// TwinCAT 3 PLC project Example
// ProgramVersion: 3.1.4022.7
// libraries:
//   LCLS Vacuum, * (SLAC - LCLS)
//   LCLSVacuumSerialDriverLib, * (SLAC - LCLS)
//   Tc2_SerialCom, * (Beckhoff Automation GmbH)
//   Tc2_Standard, * (Beckhoff Automation GmbH)
//   Tc2_System, * (Beckhoff Automation GmbH)
//   Tc3_Module, * (Beckhoff Automation GmbH)
// project tree:
//   / CommTask.TcTTO, PlcTask.TcTTO
//   GVLs/ GVL_COM.TcGVL (not stored), GVL_Devices.TcGVL
//   POUs/ MAIN.TcPOU, PRG_COM.TcPOU
// real-time tasks:
//   TASK PlcTask: cycle T#10ms, priority 20, ADS port 350
//   TASK CommTask: cycle T#10ms, priority 21, ADS port 351

CONFIGURATION Example
    RESOURCE PLC ON TwinCAT3
        TASK CommTask(INTERVAL := T#10ms, PRIORITY := 21);
        TASK PlcTask(INTERVAL := T#10ms, PRIORITY := 20);
        PROGRAM PRG_COM WITH CommTask : PRG_COM;
        PROGRAM MAIN WITH PlcTask : MAIN;
    END_RESOURCE
END_CONFIGURATION

// ---- GVLs/GVL_Devices.TcGVL
VAR_GLOBAL
	
	(*TD20*)
	{attribute 'pytmc' := '
    pv: PTM:01
	'}
	PTM_01 : FB_PTM_TurboDrive; // PLC IO Interface
	PTM_01_Serial : FB_Oerlikon_TD20_COM; //Serial Interface
	
	
	(*Pfeiffer*)
	{attribute 'pytmc' := '
    pv: PTM:02
	'}
	PTM_02 : FB_PTM_Pfeiffer;
	{attribute 'pytmc' := '
    pv: PTM:03
	'}
	PTM_03 : FB_PTM_Pfeiffer;
	// They share the same serial port
	st_Pfeiffer_CTRL 			: ARRAY[1..20] OF ST_PfeifferControl;
	st_Pfeiffer_RBK 			: ARRAY[1..20] OF ST_PfeifferStatus;
	fb_PfeifferCom : FB_PFEIFFER_COM;
	
END_VAR

// ---- POUs/PRG_COM.TcPOU
PROGRAM PRG_COM
VAR
END_VAR

//needs to run on a seperate task
//PTM_01
(*Instanitate Serial port com function *) 
fbSerialLineControl(
	Mode:= SERIALLINEMODE_EL6_22B,
	pComIn:= ADR(stComIn),
	pComOut:=ADR(stComOut),
	SizeComIn:= SIZEOF(stComIn),
	TxBuffer:= SerialTXBuffer,
	RxBuffer:= SerialRXBuffer,
	Error=> ,
	ErrorID=> );
	

//PTM_02 and PTM_03
(*Instanitate Serial port com function *) 
E2_fbSerialLineControl(
	Mode:= SERIALLINEMODE_EL6_22B,
	pComIn:= ADR(E2_stComIn),
	pComOut:=ADR(E2_stComOut),
	SizeComIn:= SIZEOF(E2_stComIn),
	TxBuffer:= E2_SerialTXBuffer,
	RxBuffer:= E2_SerialRXBuffer,
	Error=> ,
	ErrorID=> );

END_PROGRAM

// ---- POUs/MAIN.TcPOU
PROGRAM MAIN
VAR
END_VAR

	
PRG_COM();

// Leybold Turbo Drive
(* Instanitate the Function block for Pump Control*)
PTM_01(i_xExtILKOk:= TRUE , iq_stPtm=> );
(* Instanitate the Function block for serial communication with TD20 *)
PTM_01_Serial(SerialRXBuffer := SerialRXBuffer, 
				SerialTXBuffer:= SerialTXBuffer,
				astTD20Status=>);
(* Copy Status Pv's into the PTM structure*)
PTM_01.M_Serial_IO(PTM_01_Serial.astTD20Status);




//Pfeiffer Turbo
(* Instanitate the Function block for Pump Control*)
PTM_02(i_xExtIlkOK:= TRUE , iq_stPTM=> );
PTM_03(i_xExtIlkOK:= TRUE , iq_stPTM=> );

(*Assign adresses to the pfeiffer controllers connected to this serial terminal*)
st_Pfeiffer_CTRL[1].iSerialAddress :=1;
st_Pfeiffer_CTRL[1].xEnableComm := TRUE;
st_Pfeiffer_CTRL[2].iSerialAddress :=2;
st_Pfeiffer_CTRL[2].xEnableComm := TRUE;
	
(* Instanitate the Function block for serial communication with Pfeiffer*)	
fb_PfeifferCom(astPfeifferControl := st_Pfeiffer_CTRL,
			   astPfeifferStatus:= st_Pfeiffer_RBK,
				SerialRXBuffer:= E2_SerialRXBuffer,
				SerialTXBuffer:= E2_SerialTXBuffer);
				

(* Copy Status Pv's into the PTM structure*)
//PTM_02.M_Serial_IO(st_Pfeiffer_CTRL:=st_Pfeiffer_CTRL[1],st_Pfeiffer_RBK:=st_Pfeiffer_RBK[1]);
//PTM_03.M_Serial_IO(st_Pfeiffer_CTRL:=st_Pfeiffer_CTRL[2],st_Pfeiffer_RBK:=st_Pfeiffer_RBK[2]);

END_PROGRAM
